TYPE st_GPS :
STRUCT
	Latitude 	: 	REAL;
	Longitude 	: 	REAL;
	FixTime 	: 	STRING(32);
	DateTime	:	DT;
	Speed		:	REAL;
	SatCount	:	UINT;
	Accuracy	:	REAL;	
END_STRUCT
END_TYPE

(* stored: Version 1.1.0.1, ProductVersion 3.1.4026.18
   DUT st_GPS: Id {2ef5467b-5bb1-4955-b2bf-c336457b11e3} *)
